(* CODESYS project TestPlcProject.library
   Title: TestPlcProject
   Version: 0.1.0
   Placeholder: TestPlcProject
   Company: TestPlcProject

Project tree, tasks and I/O mapping:
  libraries: Tc2_Standard, * (Beckhoff Automation GmbH); Tc2_System, * (Beckhoff Automation GmbH); Tc3_Module, * (Beckhoff Automation GmbH)
  DUTs/
  GVLs/
  POUs/
    function block FB_TestFb1 [CFC]
    program MAIN [ST]
  VISUs/
*)

// POUs/FB_TestFb1
FUNCTION_BLOCK FB_TestFb1
VAR_INPUT
END_VAR
VAR_OUTPUT
END_VAR
VAR
END_VAR

END_FUNCTION_BLOCK

// POUs/MAIN
PROGRAM MAIN
VAR
END_VAR

END_PROGRAM
